TYPE StPoint :
STRUCT
    x : REAL;
    y : REAL;
END_STRUCT
END_TYPE

(* stored: Version 1.1.0.1, ProductVersion 3.1.4024.12
   DUT StPoint: Id {f4ee6c74-746c-4d39-b06e-3bb8b0d1c5e7} *)
